(* IEC 61131-3 sources: OSCAT_OpenPLC/OSCAT BASIC 3.33/OSCAT BASIC 3.33-13 String Functions/build, 2 files *)

(* ---- generated_plc.st ---- *)
FUNCTION_BLOCK BYTE_TO_STRB
  VAR_INPUT
    IN : BYTE;
    _BYTE_TO_STRB : STRING;
  END_VAR
  VAR
    i : INT;
  END_VAR

  _BYTE_TO_STRB := '';
  FOR i := 1 TO 8 DO
      IF (in AND BYTE#2#1000_0000) = BYTE#2#1000_0000 THEN
          _BYTE_TO_STRB := CONCAT(_BYTE_TO_STRB,'1');
      ELSE
          _BYTE_TO_STRB := CONCAT(_BYTE_TO_STRB,'0');
      END_IF;
  	in := SHL(in, 1);
  END_FOR;

  (* From Oscat Library, www.oscat.de *)
END_FUNCTION_BLOCK

FUNCTION_BLOCK BYTE_TO_STRH
  VAR_INPUT
    IN : BYTE;
  END_VAR
  VAR_OUTPUT
    _BYTE_TO_STRH : STRING;
  END_VAR

  _BYTE_TO_STRH:=BYTE_TO_STRING(IN,'%c');

  (* From Oscat Library, www.oscat.de *)
END_FUNCTION_BLOCK

PROGRAM program0
  VAR
    LocalVar0 : DINT;
    LocalVar1 : DINT;
    LocalVar2 : DINT;
    ADD1_OUT : DINT;
  END_VAR

  ADD1_OUT := ADD(LocalVar0, LocalVar1);
  LocalVar2 := ADD1_OUT;
END_PROGRAM

CONFIGURATION Config0

  RESOURCE Res0 ON PLC
    TASK task0(INTERVAL := T#20ms,PRIORITY := 0);
    PROGRAM instance0 WITH task0 : program0;
  END_RESOURCE
END_CONFIGURATION

(* ---- plc.st ---- *)
TYPE
  LOGLEVEL : (CRITICAL, WARNING, INFO, DEBUG) := INFO;
END_TYPE

FUNCTION_BLOCK LOGGER
  VAR_INPUT
    TRIG : BOOL;
    MSG : STRING;
    LEVEL : LOGLEVEL := INFO;
  END_VAR
  VAR
    TRIG0 : BOOL;
  END_VAR

  IF TRIG AND NOT TRIG0 THEN
  {{
   LogMessage(GetFbVar(LEVEL),(char*)GetFbVar(MSG, .body),GetFbVar(MSG, .len));
  }}
  END_IF;
  TRIG0:=TRIG;
END_FUNCTION_BLOCK

FUNCTION_BLOCK python_eval
  VAR_INPUT
    TRIG : BOOL;
    CODE : STRING;
  END_VAR
  VAR_OUTPUT
    ACK : BOOL;
    RESULT : STRING;
  END_VAR
  VAR
    STATE : DWORD;
    BUFFER : STRING;
    PREBUFFER : STRING;
    TRIGM1 : BOOL;
    TRIGGED : BOOL;
  END_VAR

  {extern void __PythonEvalFB(int, PYTHON_EVAL*);__PythonEvalFB(0, data__);}
END_FUNCTION_BLOCK

FUNCTION_BLOCK python_poll
  VAR_INPUT
    TRIG : BOOL;
    CODE : STRING;
  END_VAR
  VAR_OUTPUT
    ACK : BOOL;
    RESULT : STRING;
  END_VAR
  VAR
    STATE : DWORD;
    BUFFER : STRING;
    PREBUFFER : STRING;
    TRIGM1 : BOOL;
    TRIGGED : BOOL;
  END_VAR

  {extern void __PythonEvalFB(int, PYTHON_EVAL*);__PythonEvalFB(1,(PYTHON_EVAL*)(void*)data__);}
END_FUNCTION_BLOCK

FUNCTION_BLOCK python_gear
  VAR_INPUT
    N : UINT;
    TRIG : BOOL;
    CODE : STRING;
  END_VAR
  VAR_OUTPUT
    ACK : BOOL;
    RESULT : STRING;
  END_VAR
  VAR
    py_eval : python_eval;
    COUNTER : UINT;
    ADD10_OUT : UINT;
    EQ13_OUT : BOOL;
    SEL15_OUT : UINT;
    AND7_OUT : BOOL;
  END_VAR

  ADD10_OUT := ADD(COUNTER, 1);
  EQ13_OUT := EQ(N, ADD10_OUT);
  SEL15_OUT := SEL(EQ13_OUT, ADD10_OUT, 0);
  COUNTER := SEL15_OUT;
  AND7_OUT := AND(EQ13_OUT, TRIG);
  py_eval(TRIG := AND7_OUT, CODE := CODE);
  ACK := py_eval.ACK;
  RESULT := py_eval.RESULT;
END_FUNCTION_BLOCK

FUNCTION_BLOCK BYTE_TO_STRB
  VAR_INPUT
    IN : BYTE;
    _BYTE_TO_STRB : STRING;
  END_VAR
  VAR
    i : INT;
  END_VAR

  _BYTE_TO_STRB := '';
  FOR i := 1 TO 8 DO
      IF (in AND BYTE#2#1000_0000) = BYTE#2#1000_0000 THEN
          _BYTE_TO_STRB := CONCAT(_BYTE_TO_STRB,'1');
      ELSE
          _BYTE_TO_STRB := CONCAT(_BYTE_TO_STRB,'0');
      END_IF;
  	in := SHL(in, 1);
  END_FOR;

  (* From Oscat Library, www.oscat.de *)
END_FUNCTION_BLOCK

FUNCTION_BLOCK BYTE_TO_STRH
  VAR_INPUT
    IN : BYTE;
  END_VAR
  VAR_OUTPUT
    _BYTE_TO_STRH : STRING;
  END_VAR

  _BYTE_TO_STRH:=BYTE_TO_STRING(IN,'%c');

  (* From Oscat Library, www.oscat.de *)
END_FUNCTION_BLOCK

PROGRAM program0
  VAR
    LocalVar0 : DINT;
    LocalVar1 : DINT;
    LocalVar2 : DINT;
    ADD1_OUT : DINT;
  END_VAR

  ADD1_OUT := ADD(LocalVar0, LocalVar1);
  LocalVar2 := ADD1_OUT;
END_PROGRAM

CONFIGURATION Config0

  RESOURCE Res0 ON PLC
    TASK task0(INTERVAL := T#20ms,PRIORITY := 0);
    PROGRAM instance0 WITH task0 : program0;
  END_RESOURCE
END_CONFIGURATION
